{attribute 'qualified_only'}
VAR_GLOBAL
	//Variables for the dispensing matrix
	aDispManualValveSelection : ARRAY [1..4,1..3] OF BOOL;
	bDispTurnOnMatrix: BOOL;
	bDispResetMatrix:BOOL;
	bDispTurnOnPathing:BOOL;
	bDispActuatePath:BOOL;
	eDispStartOfPath: E_TankBundleNumber;
	eDispEndOfPath:E_OutletNumber;
	aDispStateofValves: ARRAY[1..cMaxRows,1..cMaxCols] OF E_SolenoidState;
	
	//Variables for the inlet matrix
    aInletManualValveSelection : ARRAY [1..2,1..3] OF BOOL;
	bInletTurnOnMatrix: BOOL;
	bInletResetMatrix:BOOL;
	bInbletTurnOnPathing:BOOL;
	bInletActuatePath:BOOL;
	eInletStartOfPath: E_InletToSystem;
	eInletEndOfPath:E_CompressionStages;
	aInletStateofValves: ARRAY[1..cMaxRows,1..cMaxCols] OF E_SolenoidState;
	
	//Variables for the Filling Matrix
	aFillManualValveSelection : ARRAY [1..4,1..3] OF BOOL;
	bFillTurnOnMatrix: BOOL;
	bFillResetMatrix:BOOL;
	bFillTurnOnPathing:BOOL;
	bFillActuatePath:BOOL;
	eFillStartOfPath: E_TankBundleNumber;
	eFillEndOfPath:E_CompressionStages;
	aFillStateofValves: ARRAY[1..cMaxRows,1..cMaxCols] OF E_SolenoidState;
	
	//Variables to enable and reset Sensors
	bEnableSensors:BOOL;
	bResetSensors:BOOL;
	
	//Sensor Error states
	aSensorErrors :  ARRAY[1..GVL_IO.cNumofPT] OF E_ErrorState;
	
	//Sensor Engineering values
	aPV:  ARRAY[1..GVL_IO.cNumofPT] OF REAL;
	aTV:  ARRAY[1..GVL_IO.cNumofPT] OF REAL;
	
END_VAR
VAR_GLOBAL CONSTANT
	//Set max matrix size at compile time
	cMaxRows:INT:=4;
	cMaxCols:INT:=3;
END_VAR

(* stored: Version 1.1.0.1
   GVL GVL_HMI: Id {6588a7f2-21fd-4376-97e1-41ec9d8aa579} *)
